TYPE ST_3DPoint :
STRUCT
	X : REAL; //X Koordinate in µm
	Y : REAL; //Y Koordinate in µm
	Z : REAL; //Z Koordinate in µm
END_STRUCT
END_TYPE

(* stored: Version 1.1.0.1, ProductVersion 3.1.0.23
   DUT ST_3DPoint: Id {9335b17c-d459-497d-b2cd-5c065cb6b5c6} *)
